Staubli VAL3: onStop.pgx

public program onStop(string& x_sItem[])
begin
  //
  // Done after a stop
  //
end
